FUNCTION_BLOCK PACK_WORD (* Packs 16 BOOLs into a WORD *)
  (* Standard: 61499-1; Classification: Math *)
  (* Version 0.1, 2002-05-07, JHC, Rockwell Automation, Changed SD_x to INx. *)
  (* Version 0.0, 2002-05-01, JHC, Rockwell Automation, Copied/Modified from PUBLISH_4 *)
  (* Compiler header: package fb.rt.math; *)
  (* Compiler Java IBM VisualAge 3.0 *)
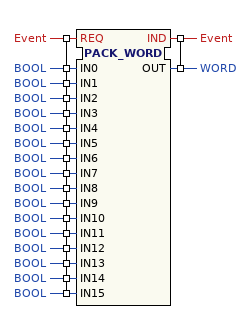
  EVENT_INPUT
    REQ WITH IN0, IN1, IN2, IN3, IN4, IN5, IN6, IN7, IN8, IN9, IN10, IN11, IN12, IN13, IN14, IN15; (* Pack Request *)
  END_EVENT
  EVENT_OUTPUT
    IND WITH OUT; (* Data Change Notification *)
  END_EVENT
  VAR_INPUT
    IN0 : BOOL; (* Data to Pack *)
    IN1 : BOOL;
    IN2 : BOOL;
    IN3 : BOOL;
    IN4 : BOOL;
    IN5 : BOOL;
    IN6 : BOOL;
    IN7 : BOOL;
    IN8 : BOOL;
    IN9 : BOOL;
    IN10 : BOOL;
    IN11 : BOOL;
    IN12 : BOOL;
    IN13 : BOOL;
    IN14 : BOOL;
    IN15 : BOOL;
  END_VAR
  VAR_OUTPUT
    OUT : WORD; (* Packed Data *)
  END_VAR
  SERVICE APPLICATION/PACK_WORD
    SEQUENCE dataChanged
      APPLICATION.REQ(IN0,...,IN15) -> PACK_WORD.pack() -> APPLICATION.IND(OUT);
    END_SEQUENCE
    SEQUENCE dataUnchanged
      APPLICATION.REQ(IN0,...,IN15) -> PACK_WORD.pack();
    END_SEQUENCE
  END_SERVICE
END_FUNCTION_BLOCK
